{region '#Template'}
	{attribute 'Version' := '5.1.0.0'}
	{attribute 'Tags' := '"LCID": "1031", "Text": "RA, Sensoren, DALI, Präsenzmelder"'}
	{attribute 'Tags' := '"LCID": "1033", "Text": "RA, Sensors, DALI, presence-detection"'}
	{attribute 'Description' := '"LCID": "1031", "Text": "Template DALI Präsenzmelder"'}
	{attribute 'Description' := '"LCID": "1033", "Text": "Template DALI presence-detection"'}
{endregion}
FUNCTION_BLOCK FB_BA_BrightnessPresenceDALI EXTENDS FB_BA_Ext_BrightnessPresence_Base

VAR_INPUT
	bEn						: BOOL;			// FB-enable
	bInitialize				: BOOL;			// initialize with DALI-parameters
	bResetPresence			: BOOL;			// reset internal PLC-programmed delay-timer and trigger bRstSwi
	{attribute 'parameterUnit':= 's'}
	nPrdQueryBrtns			: UDINT	:= 1;	// [s] query interval of brightness
END_VAR
VAR_OUTPUT
	bPresence				: BOOL;			// presence detected
	bPresenceDelayActive	: BOOL;			// presence detection is FALSE, output bPresence is only set by delay-timer 
	bRstSwi					: BOOL;			// reset manual switch especially for sunblinds (presence for sunblinds differs between thermoautomatic and sunprotection)
	fBrightness				: REAL;			// brightness value
	bInitializing			: BOOL;			// device is being initialized
	bErr					: BOOL;			// error
END_VAR
VAR_INPUT CONSTANT PERSISTENT
	nAdr					: BYTE;	
	nInstancePresence		: BYTE;	
	nInstanceBrightness		: BYTE;	
	nResBrtns				: BYTE;			// manufacturers specific resolution	
	ipDALICommunication		: Tc3_DALI.I_DALICommunication;
END_VAR
VAR_INPUT CONSTANT
	BrightnessPresenceSns	: FB_BA_BrtnsPrcDALI;
	PresenceDelay			: FB_BA_PresenceMonitoring;		
	Brightness				: FB_BA_AI_Raw;
	Presence				: FB_BA_BI_Raw;		
END_VAR
VAR
END_VAR

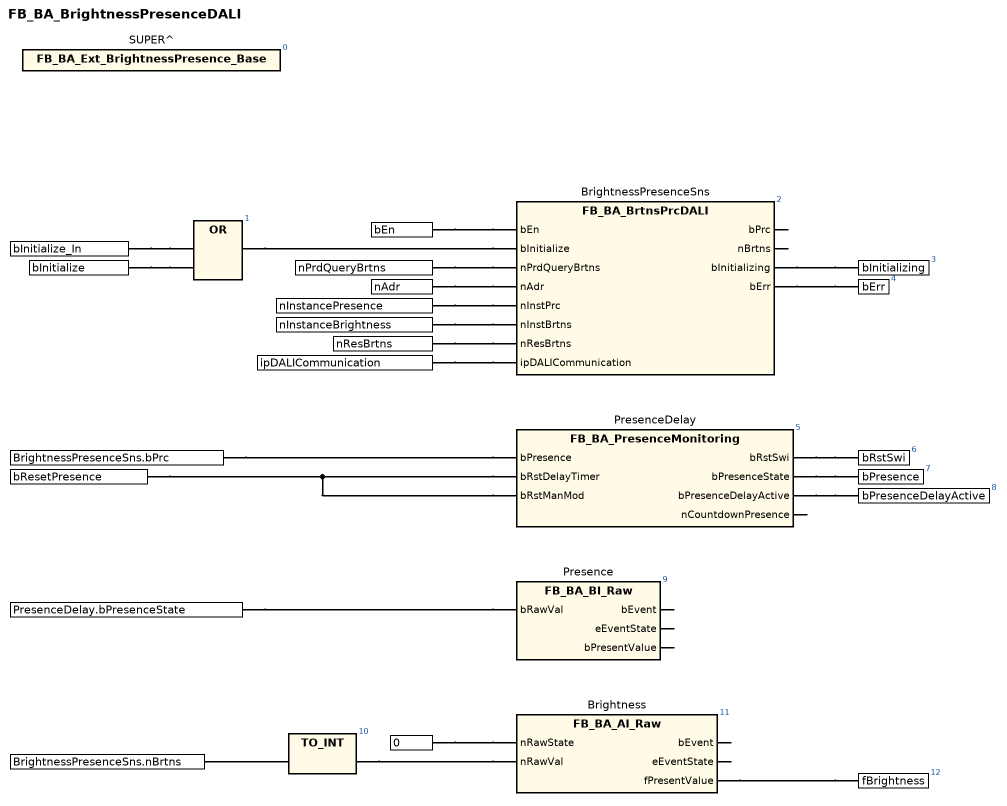
SUPER^(); // FB_BA_Ext_BrightnessPresence_Base
BrightnessPresenceSns(
    bEn := bEn,
    bInitialize := bInitialize_In OR bInitialize,
    nPrdQueryBrtns := nPrdQueryBrtns,
    nAdr := nAdr,
    nInstPrc := nInstancePresence,
    nInstBrtns := nInstanceBrightness,
    nResBrtns := nResBrtns,
    ipDALICommunication := ipDALICommunication); // FB_BA_BrtnsPrcDALI
bInitializing := BrightnessPresenceSns.bInitializing;
bErr := BrightnessPresenceSns.bErr;
PresenceDelay(
    bPresence := BrightnessPresenceSns.bPrc,
    bRstDelayTimer := bResetPresence,
    bRstManMod := bResetPresence); // FB_BA_PresenceMonitoring
bRstSwi := PresenceDelay.bRstSwi;
bPresence := PresenceDelay.bPresenceState;
bPresenceDelayActive := PresenceDelay.bPresenceDelayActive;
Presence(bRawVal := PresenceDelay.bPresenceState); // FB_BA_BI_Raw
Brightness(nRawState := 0, nRawVal := TO_INT(BrightnessPresenceSns.nBrtns)); // FB_BA_AI_Raw
fBrightness := Brightness.fPresentValue;

METHOD FB_init : BOOL
VAR_INPUT
	bInitRetains : BOOL; // if TRUE; the retain variables are initialized (warm start / cold start)
	bInCopyCode : BOOL;  // if TRUE; the instance afterwards gets moved into the copy code (online change)
END_VAR
BrightnessPresenceSns.nDeadtime			:= 2;				// Dead-time-timer as multiple of 50ms
BrightnessPresenceSns.nHold				:= 5;				// Hold-timer as multiple of 10s, a "0" means 1s
BrightnessPresenceSns.nReport			:= 60;				// Report-timer in s BrightnesPresenceSns

PresenceDelay.nDlyPrc					:= 600;				// Presence delay [s] (in addition to the DALI-hold-timer!)			
	
// Presence-detection (delayed) // Präsenzmeldung ausschaltverzögert	
Presence.iParent						:= THIS^;								
Presence.iLabel							:= LblFun_Status;
Presence.ePolarity						:= E_BA_Polarity.eNormal;
Presence.sActiveText 					:= txtEvent_Occupied;
Presence.sInactiveText 					:= txtEvent_NotOccupied;
Presence.nEventClassID					:= EC_ID.NC80;
Presence.stTimeDelay.nToNormal			:= 0;
Presence.stTimeDelay.nToAbnormal		:= 0;
Presence.bAlarmValue					:= TRUE;
Presence.aEventTransitionText[1]		:= txtEvent_Triggered;
Presence.aEventTransitionText[2]		:= txtEvent_Error;
Presence.aEventTransitionText[3]		:= txtEvent_Normal;
Presence.bEventDetectionEnable			:= TRUE;
Presence.eEnPlantLock					:= E_BA_LockPriority.eNoLock;

// Brightness scaled // skalierte Helligkeit
Brightness.iParent						:= THIS^;		
Brightness.iLabel						:= LblFun_MeasuredValue;
Brightness.eUnit						:= E_BA_Unit.eLight_Luxes;
Brightness.fResolution 					:= 1; // in case, the manufacturer supplies a lux-value
Brightness.fScaleOffset 				:= 0; 	
Brightness.fCOVIncrement				:= BA2_Param.fDefCOVIncrement;
Brightness.nEventClassID				:= EC_ID.NC80;
Brightness.stTimeDelay.nToNormal		:= BA2_Param.nDefTimeDelay_ToNormal;
Brightness.stTimeDelay.nToAbnormal		:= BA2_Param.nDefTimeDelay_ToAbnormal;
Brightness.stHighLimit.bEnable			:= FALSE;
Brightness.stHighLimit.fValue			:= 0.0;		
Brightness.stLowLimit.bEnable			:= FALSE;
Brightness.stLowLimit.fValue			:= 0.0;
Brightness.fLimitDeadband 				:= BA2_Param.fDefLimitDeadband;
Brightness.aEventTransitionText[1]		:= txtEvent_Exceeded;
Brightness.aEventTransitionText[2]		:= txtEvent_Disturb;
Brightness.aEventTransitionText[3]		:= txtEvent_Normal;
Brightness.bEventDetectionEnable		:= TRUE;
Brightness.eEnPlantLock					:= E_BA_LockPriority.eNoLock;
END_METHOD

END_FUNCTION_BLOCK

(* stored: Version 1.1.0.1, ProductVersion 3.1.4024.12
   POU FB_BA_BrightnessPresenceDALI: Id {cea76f88-7ba1-40ec-a113-1bc3965656b1}, SpecialFunc None
   Method FB_init: Id {ecf11d18-8015-41b5-a072-5fdd9640e40a} *)
